# EPICS substitutions: ipimbLib/Db/ipimbTpr.substitutions
file ipimbCH.tpl-db
{
    pattern
    { CHANNEL    DONECTR }
    { 0,         "$(RECNAME):DONE_CNT.A" }
    { 1,         "$(RECNAME):DONE_CNT.B" }
    { 2,         "$(RECNAME):DONE_CNT.C" }
    { 3,         "$(RECNAME):DONE_CNT.D" }
}

file ipimbALL.tpl-db
{
    { IOC = $(IOC), GETFIDFUNC = ipimbGetFiducial, TRIGEN = $(TPR):CH$(TRIG)_SYS0_TCTL }
}

file ipimbSyncTpr.tpl-db
{
    { IOC = $(IOC) }
}
